TYPE ST_ITC_GCR :
(**************************************************************************************
 * 	Application		:	BoxControl Framework
 *	Revision		:	$Revision: 404529 $
 *	Revision date	:	$Date: 2018-04-23 08:21:38 +0200 (Mo., 23 Apr 2018) $
 *	Last changed by	:	$Author: b7bolm $
 *	URL				:	$URL: http://almscdc.swisslog.com/repo/SWPD/Development/BoxControlFramework/20_Release/trunk/01_Software/BCF/BCF/JumpStart/20_Product/10_App/11_Com/10_Lib/10_Conv/11_ITC/01_DUTs/ST_ITC_GCR.TcDUT $
 *
 *	Purpose			:	GCR Structure
 *
 * ------------------------------------------------------------------------------------
 *	Copyright Swisslog [IP AG], Switzerland. All rights reserved.
 * 
 * ------------------------------------------------------------------------------------
 *	
 * 	Revision History: 
 *
 * 	VERSION			DATE			INITIALS			DESCRIPTION
 *	0.1				01.01.2001		swl					Example
 *
 **************************************************************************************)
STRUCT
	GroupName		: STRING(Conveyor.POSITION_STRINGLENGTH); // 12 Digit SIS Group Name MM-GGG-0000-000 
	Code			: INT; // 2 Digit Control code 
	Variable		: DINT; // 4 DigitControl code variable 
	ReturnCode		: E_ErrorConv; // 4 Digit Return Code 
END_STRUCT
END_TYPE

(* stored: Version 1.1.0.1, ProductVersion 3.1.4022.12
   DUT ST_ITC_GCR: Id {9cdf3fa4-1295-40af-a618-e2e5a6dba275} *)
